Fanuc KAREL source: kt00303.KL

PROGRAM KT00303
%STACKSIZE=65535
%PRIORITY=65535
%NOLOCKGROUP
VAR
I2 : INTEGER
OUT : BOOLEAN
-- UNRESOLVED DECLARATIONS (source type spelling not recovered)
-- Y1 : ARRAY[2] OF TYPE_0x0018 (type_u16=0x2018)
BEGIN
Y1[1]=2
I2=3
-- UNRESOLVED_PC line 10 opcodes [22 9D 33 B1 21 58 23] marker_code=35
END KT00303
